SYSTEM test_Training_06_OPC_UA
  (* Version 1.0, 2026-09-04, Franz Höpfinger, Meisterschulen am Ostbahnhof *)
  PACKAGE Training_OPC_UA_RES5;
  IMPORT logiBUS::stations::Computers::C_11;
  IMPORT logiBUS::stations::Computers::C_12;
  APPLICATION App_OPC_UA_RES5
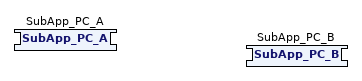
    SUBAPPS
      SubApp_PC_A : subapp::Training_06_OPC_UA_RES::SubApp_PC_A;
      SubApp_PC_B : subapp::Training_06_OPC_UA_RES::SubApp_PC_B;
    END_SUBAPPS
  END_APPLICATION
  DEVICE FORTE_PC_A : iec61499::system::FORTE_PC(MGR_ID := C_11 (* Device manager socket ID *))
    {SET_ATTRIBUTE(Profile, HOLOBLOC)}
    RESOURCE EMB_RES_A : iec61499::system::EMB_RES
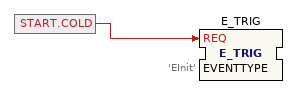
      FBS
        E_TRIG : iec61499::events::E_TRIG(EVENTTYPE := 'EInit');
      END_FBS
      EVENT_CONNECTIONS
        START.COLD TO E_TRIG.REQ;
      END_CONNECTIONS
    END_RESOURCE
  END_DEVICE
  DEVICE FORTE_PC_B : iec61499::system::FORTE_PC(MGR_ID := C_12 (* Device manager socket ID *))
    {SET_ATTRIBUTE(Profile, HOLOBLOC)}
    RESOURCE EMB_RES_B : iec61499::system::EMB_RES
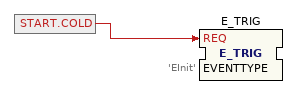
      FBS
        E_TRIG : iec61499::events::E_TRIG(EVENTTYPE := 'EInit');
      END_FBS
      EVENT_CONNECTIONS
        START.COLD TO E_TRIG.REQ;
      END_CONNECTIONS
    END_RESOURCE
  END_DEVICE
  MAPPINGS
    App_OPC_UA_RES5.SubApp_PC_A ON FORTE_PC_A.EMB_RES_A;
    App_OPC_UA_RES5.SubApp_PC_B ON FORTE_PC_B.EMB_RES_B;
  END_MAPPINGS
  SEGMENTS
    Ethernet : iec61499::system::Ethernet;
  END_SEGMENTS
  LINKS
    FORTE_PC_A => Ethernet;
    FORTE_PC_B => Ethernet;
  END_LINKS
END_SYSTEM
